// TwinCAT 3 PLC project Piper
// ProgramVersion: 3.1.4024.0
// libraries:
//   Tc2_Standard, * (Beckhoff Automation GmbH)
//   Tc2_System, * (Beckhoff Automation GmbH)
//   Tc3_Module, * (Beckhoff Automation GmbH)
// project tree:
//   Piper/1_Controller/ Piper.TcPOU (not stored), PiperCommand.TcDUT, PiperStatus.TcDUT (not stored), PiperSubmoduleCollection.TcDUT (not stored), PIPER_CONST.TcGVL (not stored)
//   Piper/2_Plugin/ IPiperModule.TcIO (not stored), PiperImplements.TcDUT (not stored), PiperModule.TcPOU (not stored), PiperModuleInternal.TcDUT (not stored)
//   Piper/3_Context/ PiperNullContext.TcPOU (not stored)
//   Piper/4_Utilities/ GroupStatus.TcPOU
//   / PlcTask.TcTTO (not stored)
//   POUs/ MAIN.TcPOU
// real-time tasks:
//   TASK PlcTask: cycle T#10ms, priority 20, ADS port 350

// ---- Piper/1_Controller/PiperCommand.TcDUT
TYPE PiperCommand :
STRUCT
	Abort : BOOL;
	Start : BOOL;
	Stop : BOOL;
	Clear : BOOL;
	Reset : BOOL;
	Suspend : BOOL;
	Unsuspend : BOOL;
	Hold : BOOL;
	Unhold : BOOL;
END_STRUCT
END_TYPE;

// ---- Piper/4_Utilities/GroupStatus.TcPOU
FUNCTION_BLOCK GroupStatus
VAR_INPUT
END_VAR
VAR_OUTPUT
END_VAR
VAR
	_Busy : BOOL;
	_Error : BOOL;	
END_VAR

METHOD Busy
VAR_INPUT
	Message : STRING[80];
END_VAR
_Busy := TRUE;
END_METHOD

METHOD Error
VAR_INPUT
	Message : STRING[80];
END_VAR
_Error := TRUE;
END_METHOD

PROPERTY isBusy : BOOL
GET
isBusy := NOT _Error AND _Busy;
END_GET
END_PROPERTY

PROPERTY isDone : BOOL
GET
isDone := NOT _Error AND NOT _Busy;
END_GET
END_PROPERTY

PROPERTY isError : BOOL
GET
isError := _Error;
END_GET
END_PROPERTY

METHOD Ok : BOOL
VAR_INPUT
END_VAR
END_METHOD

METHOD Reset
VAR_INPUT
END_VAR
_Busy := FALSE;
_Error := FALSE;
END_METHOD

PROPERTY status : PLCOpenStatusBase
GET
IF _Error THEN
	
status := PLCOpenStatusBase.ERROR;

ELSIF _Busy THEN

status := PLCOpenStatusBase.BUSY;

ELSE

status := PLCOpenStatusBase.ERR_OK;
	
END_IF
END_GET
END_PROPERTY

END_FUNCTION_BLOCK

// ---- POUs/MAIN.TcPOU
PROGRAM MAIN
VAR
END_VAR

END_PROGRAM
